RoboDK station: robot_base.rdk

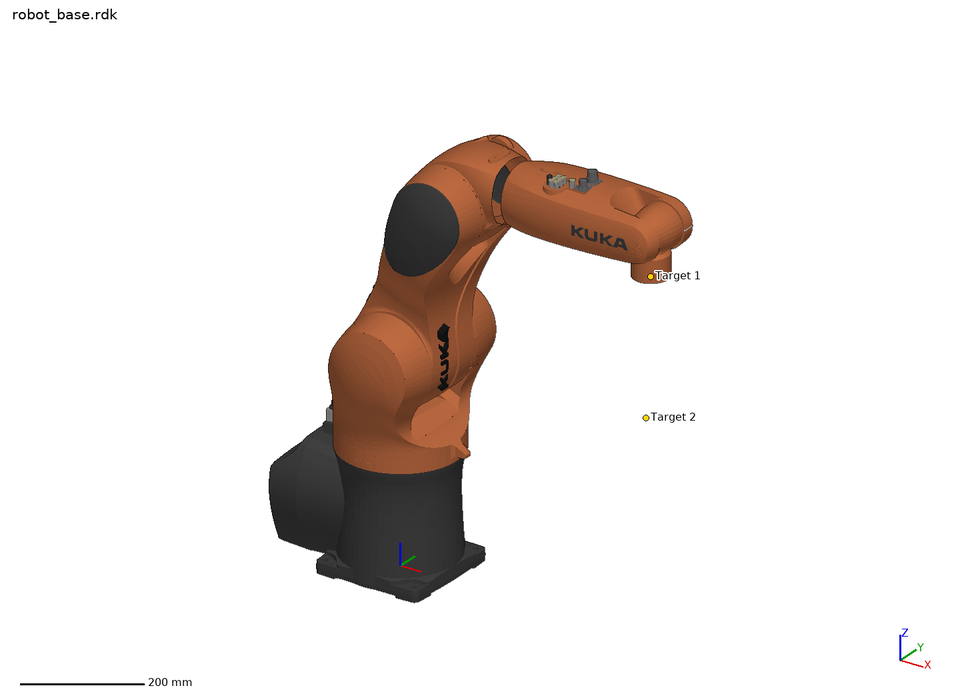
[picture v0: the station drawn from its stored meshes, robots at their saved joint values, targets as dots, program paths as lines]
Station robot_base (saved by RoboDK 5.3.0). Poses are relative to the parent item; angles as X-Y-Z fixed-axis rotations.
  - frame KUKA KR 6 R700 sixx Base at (0, 0, 0) mm
    - robot KUKA KR 6 R700 sixx: 6 axes, payload 6 kg, reach 706.7 mm, repeatability 0.03 mm, weight 50 kg
        modified DH rows (alpha deg, a mm, theta deg, d mm): 0, 0, 0, 400; -90, 25, 0, 0; 0, 315, -90, 0; -90, 35, 0, 365; 90, 0, 0, 0; -90, 0, 180, 80
        joint limits [-170, -190, -120, -185, -120, -350] to [170, 45, 156, 185, 120, 350]; home [0, -90, 90, 0, 0, 0]; saved at [0, -70.995, 70.557, 0, 90.437, 0]
    - target Target 1 (Cartesian target) at (492.3, 0, 655.61) mm, rotated rx 180 ry 0 rz -180 deg; joints [0, -70.995, 70.557, 0, 90.437, 0] of KUKA KR 6 R700 sixx
    - target Target 2 (Cartesian target) at (483.17, 0, 399.18) mm, rotated rx -180 ry 0 rz -180 deg; joints [0, -61.65, 99.818, 0, 51.832, 0] of KUKA KR 6 R700 sixx
